FUNCTION_BLOCK Door_Controller (* Composite Function Block Type *)
  (* Standard: 61499-2 *)
  (* Version 0.0, 9/24/2026, macie, Schneider Electric, template *)
  PACKAGE Main;
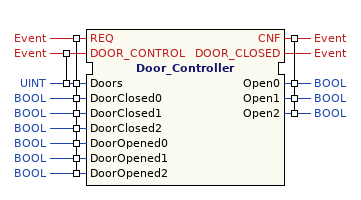
  EVENT_INPUT
    REQ WITH Doors, DoorOpened0, DoorClosed0, DoorOpened1, DoorClosed1, DoorOpened2, DoorClosed2; (* Normal Execution Request *)
    DOOR_CONTROL WITH Doors;
  END_EVENT
  EVENT_OUTPUT
    CNF WITH Open0, Open1, Open2; (* Execution Confirmation *)
    DOOR_CLOSED;
  END_EVENT
  VAR_INPUT
    Doors : UINT; (* Input event qualifier *)
    DoorClosed0 : BOOL;
    DoorClosed1 : BOOL;
    DoorClosed2 : BOOL;
    DoorOpened0 : BOOL;
    DoorOpened1 : BOOL;
    DoorOpened2 : BOOL;
  END_VAR
  VAR_OUTPUT
    Open0 : BOOL; (* Output event qualifier *)
    Open1 : BOOL;
    Open2 : BOOL;
  END_VAR
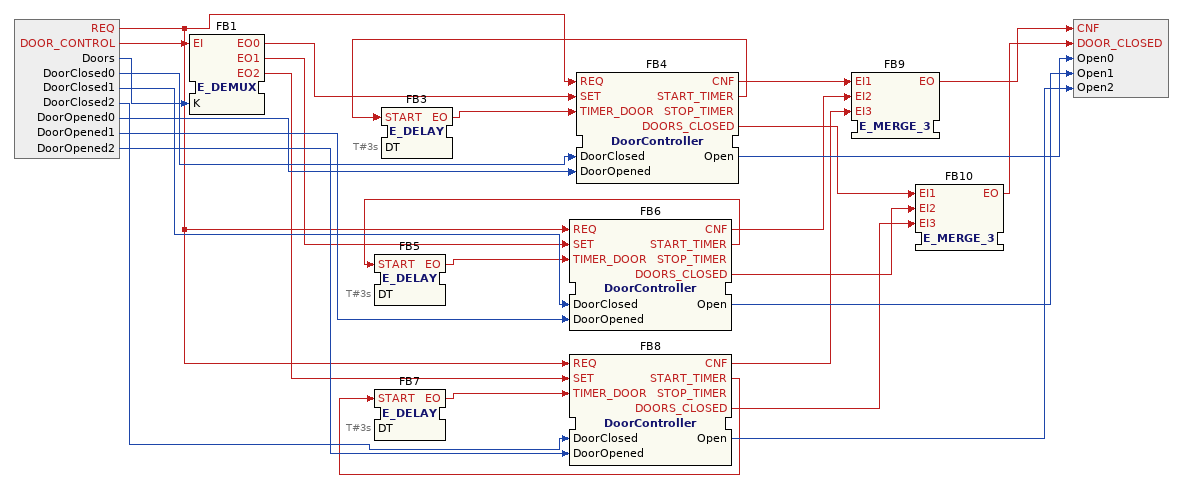
  FBS
    FB1 : E_DEMUX;
    FB3 : E_DELAY(DT := T#3s);
    FB4 : DoorController;
    FB5 : E_DELAY(DT := T#3s);
    FB6 : DoorController;
    FB7 : E_DELAY(DT := T#3s);
    FB8 : DoorController;
    FB9 : E_MERGE_3;
    FB10 : E_MERGE_3;
  END_FBS
  EVENT_CONNECTIONS
    FB1.EO0 TO FB4.SET;
    FB3.EO TO FB4.TIMER_DOOR;
    FB4.START_TIMER TO FB3.START;
    FB5.EO TO FB6.TIMER_DOOR;
    FB6.START_TIMER TO FB5.START;
    FB7.EO TO FB8.TIMER_DOOR;
    FB8.START_TIMER TO FB7.START;
    FB1.EO1 TO FB6.SET;
    FB1.EO2 TO FB8.SET;
    FB9.EO TO CNF;
    FB4.CNF TO FB9.EI1;
    FB6.CNF TO FB9.EI2;
    FB8.CNF TO FB9.EI3;
    DOOR_CONTROL TO FB1.EI;
    REQ TO FB4.REQ;
    REQ TO FB6.REQ;
    REQ TO FB8.REQ;
    FB4.DOORS_CLOSED TO FB10.EI1;
    FB6.DOORS_CLOSED TO FB10.EI2;
    FB8.DOORS_CLOSED TO FB10.EI3;
    FB10.EO TO DOOR_CLOSED;
  END_CONNECTIONS
  DATA_CONNECTIONS
    Doors TO FB1.K;
    DoorOpened0 TO FB4.DoorOpened;
    DoorClosed0 TO FB4.DoorClosed;
    FB4.Open TO Open0;
    FB6.Open TO Open1;
    FB8.Open TO Open2;
    DoorClosed2 TO FB8.DoorClosed;
    DoorOpened2 TO FB8.DoorOpened;
    DoorOpened1 TO FB6.DoorOpened;
    DoorClosed1 TO FB6.DoorClosed;
  END_CONNECTIONS
END_FUNCTION_BLOCK
